// TIA Portal V16 export
// export: Created 2021-07-12T14:47:20.1467383Z, ExportSetting WithDefaults, DisplayName Totally Integrated Automation Portal, DisplayVersion V16, DisplayName TIA Portal Version Control Interface, DisplayVersion V16, DisplayName TIA Portal Openness, DisplayVersion V16, DisplayName STEP 7 Professional, DisplayVersion V16, DisplayName STEP 7 Safety, DisplayVersion V16, DisplayName WinCC Professional, DisplayVersion V16
TYPE "SimaHydTO_typeHMIConnectionBasicAxisControlStatus"
TITLE = SimaHydTO_typeHMIConnectionBasicAxisControlStatus
// HMI interface: Basic axis control (LAxisBasics) - Status (PLC -> HMI)
// stored: IsFailsafeCompliant false
   STRUCT
      powerStatus : Bool;   // MC_Power: 0: Technology object disabled / 1: Technology object enabled
      powerBusy : Bool;   // MC_Power: Job is running
      resetDone : Bool;   // MC_Reset: Error has been acknowledged or Restart has been executed.
      resetBusy : Bool;   // MC_Reset: Job is running
      resetFBDone : Bool;   // LSimaHyd_MC_Reset: Error has been acknowledged or Restart has been executed.
      resetFBBusy : Bool;   // LSimaHyd_MC_Reset: Job is running
      homeDone : Bool;   // MC_Home: Job is completed
      homeBusy : Bool;   // MC_Home: Job is running
      jogInVelocity : Bool;   // MC_MoveJog: The velocity setpoint / speed setpoint was reached and will be maintained
      jogBusy : Bool;   // MC_MoveJog: Job is running
      commandAborted : Bool;   // The job was aborted by another job during execution (see also StatusID)
      error : Bool;   // An error occurred during execution of the job. The job is rejected. The cause of the error can be found in the "ErrorID" parameter.
      errorID : Word;   // ErrorID of motion control instruction (see also StatusID)
      statusID : Int;   // Additional specification of affected Motion control instruction of CommandAborted or Error: 0: No instruction / 1: MC_Power / 2: MC_Reset / 3: MC_Home / 4: MC_MoveJog
   END_STRUCT;
END_TYPE
